// TIA Portal V20 export
// export: Created 2025-12-01T14:57:03.8292158Z, ExportSetting None, DisplayName Totally Integrated Automation Portal, DisplayVersion V20 Update 3, DisplayName TIA Portal Openness, DisplayVersion V20 Update 3, DisplayName TIA Portal Version Control Interface, DisplayVersion V20 Update 3, DisplayName STEP 7 Professional, DisplayVersion V20 Update 3, DisplayName STEP 7 Safety, DisplayVersion V20 Update 2, DisplayName WinCC Basic/Comfort/Advanced, DisplayVersion V20 Update 3, DisplayName WinCC Professional, DisplayVersion V20 Update 3, DisplayName WinCC Unified, DisplayVersion V20 Update 3
FUNCTION "FC702_JDT02RecJdTMensaje" : Void   // FC702, LAD
TITLE = "RecJdTMensaje" Recepción del Mensaje enviado por TCP/IP
{ S7_Optimized_Access := 'FALSE' }
AUTHOR : TRACKING
NAME : 20141014
VERSION : 4.0
// Pasos a seguir, por orden
// 
// - Recoger cabecera
// - Recoger cuerpo
// - Transferir Mensaje recibido por TCP/IP
// stored: AutoNumber false, SetENOAutomatically false
   VAR_TEMP
      DBRecJdt : Word;   // DB de Recpcion de Mensaje
      DBUltimoRec : Word;   // DB del Ultimo Mensaje Recibido
      Longitud : UDInt;   // Longitud del cuerpo
      CantidadBytes : UDInt;   // Cantidad de Bytes de los Eventos
      RecJdT_Longitud : UDInt;   // Longitud de Bytes que recibe en AG_RECV
      ReturnValor : Int;   // Temporal
      POrigen : Any;   // Puntero ANY del Origen
      PDestino : Any;   // Puntero ANY del Destino
   END_VAR
BEGIN

NETWORK
TITLE = Inicializaciones
// -------------------------------------------------------------------------------------------
// Si trabaja sin Agencia  2018 01 24
      SET;
      AN    "Activar_JDT02";  // Mirar si se trabaja con agencia
      JC    Final;

// ------------------------------------------------------------------------------------------------------
// Inicializamos las variables de los DB
      L     "JDT2_NDB_RecMensaje";  // Cogemos el Numero del DB de RecepMensaje
      T     #DBRecJdt;
      L     "JDT2_NDB_UltimoRec";  // Cogemos el Numero del DB de UltimoRecibido
      T     #DBUltimoRec;

// ------------------------------------------------------------------------------------------------------
// Comprobamos el EnlaceCP
      AN    "DB701_JDT02StatusCOM".EnlaceCP_OK;  // Mirar Si esta el EnlaceCP Activo
      JCN   Inicio;

      R     "DB701_JDT02StatusCOM".RecJdT_Cabecera;  // Resetear Variables
      R     "DB701_JDT02StatusCOM".RecJdT_Cuerpo;

      CALL  "FC898_BorrarMensaje"
      ( DB_A_RESET := "DB702_JDT02RecepMensaje"  // ¿Hay que borrarlo?
      );

      JU    Final;  // Finalizar


NETWORK
TITLE = Distribucion
// Orden a mirar para distribucion del trabajo
// - Esta el Cuerpo recogida - Transferir
// - Esta la cabecera recogida - Recoger el Cuerpo
// - Recoger la Cabecera
Inicio:NOP   0;
      SET;
      A     "DB701_JDT02StatusCOM".RecJdT_Cuerpo;  // Esta recogido el Cuerpo
      JC    TranferirMensaje;  // Ir a Transferir el Mensaje

      A     "DB701_JDT02StatusCOM".RecJdT_Cabecera;  // Esta recogido la Cabecera
      JC    RecogerCuerpo;  // Ir a Recoger el Cuerpo

      JU    RecogerCabeza;  // Ir a Recoger la Cabecera



NETWORK
TITLE = Recepcion de la Cabeza del Mensaje
// Pasos a seguir:
// - Generar el Punterp para recoger la Cabecera
// - Mirar si ha llegado la cabecera
// - Comprobación del mensaje recibido es correcto
// - Mirar si hay que resetear el Enlace
// -----------------------------------------------------------------------------------------------------
// 1º Paso - Generar el Puntero para recoger la Cabecera

RecogerCabeza:CALL  "FC897_Generar_PointerAny"
      ( TYP           := 16#10,
        DataTyp       := 16#02,
        repeatcounter := 22,  // Tamaño de la cabecera
        DB_Number     := "JDT2_NDB_RecMensaje",  // DB donde guardar la cabecera
        storearea     := 16#84,
        storeaddresse := 16#0000_0000,
        Any_Pointer   := #POrigen  // Puntero de la cabecera
      );

// -----------------------------------------------------------------------------------------------------
// 2º Paso - Mirar si la llegado la cabecera

      AN    "DB891_VariablesTCP".TRCV_JdT_PLC_Req_JDT02;
      AN    "DB891_VariablesTCP".TRCV_JdT_PLC_Busy_JDT02;
      S     "DB891_VariablesTCP".TRCV_JdT_PLC_Req_JDT02;

      CALL  TRCV, "DB899_TRCV_JdT_PLC_JDT02"
      ( EN_R     := "DB891_VariablesTCP".TRCV_JdT_PLC_Req_JDT02,
        ID       := W#16#3,
        LEN      := 22,
        ADHOC    := ,
        NDR      := "DB891_VariablesTCP".TRCV_JdT_PLC_Done_JDT02,
        BUSY     := "DB891_VariablesTCP".TRCV_JdT_PLC_Busy_JDT02,
        ERROR    := "DB891_VariablesTCP".TRCV_JdT_PLC_Error_JDT02,
        STATUS   := "DB891_VariablesTCP".TRCV_JdT_PLC_Status_JDT02,
        RCVD_LEN := #RecJdT_Longitud,
        DATA     := #POrigen
      );



// -----------------------------------------------------------------------------------------------------
// 3º Paso - Comprobación del mensaje recibido

      A     "DB891_VariablesTCP".TRCV_JdT_PLC_Req_JDT02;  // Si llega el Inicio de Mensaje 0x02
      A     "DB891_VariablesTCP".TRCV_JdT_PLC_Done_JDT02;  // Cabecera ya recogida
      AN    "DB891_VariablesTCP".TRCV_JdT_PLC_Error_JDT02;
      A(;
      L     "DB702_JDT02RecepMensaje".Mensaje[0];
      L     2;
      ==I;
      );
      S     "DB701_JDT02StatusCOM".RecJdT_Cabecera;
      R     "DB891_VariablesTCP".TRCV_JdT_PLC_Req_JDT02;



// -----------------------------------------------------------------------------------------------------
// 4º Paso - Hay que resetear el Enlace

      A     "DB891_VariablesTCP".TRCV_JdT_PLC_Req_JDT02;  // Sino llega el Inicio de Mensaje 0x02
      A     "DB891_VariablesTCP".TRCV_JdT_PLC_Done_JDT02;  // Resetear
      AN    "DB891_VariablesTCP".TRCV_JdT_PLC_Error_JDT02;
      A(;
      L     "DB702_JDT02RecepMensaje".Mensaje[0];
      L     2;
      <>I;
      );
      S     "DB701_JDT02StatusCOM".RecJdT_Reset;
      R     "DB891_VariablesTCP".TRCV_JdT_PLC_Req_JDT02;

      A     "DB891_VariablesTCP".TRCV_JdT_PLC_Req_JDT02;  //Si llega Error en la Recepcio
      AN    "DB891_VariablesTCP".TRCV_JdT_PLC_Done_JDT02;  // Resetear
      A     "DB891_VariablesTCP".TRCV_JdT_PLC_Error_JDT02;
      S     "DB701_JDT02StatusCOM".RecJdT_Reset;
      R     "DB891_VariablesTCP".TRCV_JdT_PLC_Req_JDT02;


//////////////////////////////////////////////////////////////////////////
/// Final (Alonso) 2019 09 19
      SET;
      A     "DB701_JDT02StatusCOM".RecJdT_Cabecera;
      JC    RecogerCuerpo;

      JU    Final;  // Finalizar



NETWORK
TITLE = Recepcion del Cuerpo del Mensaje
// Pasos a seguir
// - Conseguir la longitud del cuerpo
// - Generar el puntero para recoger el cuerpo
// - Mirar si ha llegado el cuerpo
// - Comprobación del mensaje recibido es correcto
// - Mirar si hay que resetear el Enlace
// -----------------------------------------------------------------------------------------------------
// 1º Paso - Conseguir la longitud del cuerpo
RecogerCuerpo:CALL  "FC890_EtiqChar_EtiqDInt"
      ( DB_String   := "JDT2_NDB_RecMensaje",
        Long_String := 5,
        Offset_Ini  := 20,
        Valor       := #Longitud
      );  // Conseguir del Mensaje su longitud

      L     #Longitud;
      T     "DB701_JDT02StatusCOM".RecJdT_LongitudCuerpo;  // Guardo la longitud del Mensaje

      L     "DB701_JDT02StatusCOM".RecJdT_LongitudCuerpo;  // Calculo la longitud del Cuerpo
      L     22;
      -I;
      T     #CantidadBytes;


// -----------------------------------------------------------------------------------------------------
// 2º Paso - Generar el Puntero para recoger la Cuerpo
      CALL  "FC897_Generar_PointerAny"
      ( TYP           := 16#10,
        DataTyp       := 16#02,
        repeatcounter := #CantidadBytes,  // Tamaño del cuerpo
        DB_Number     := "JDT2_NDB_RecMensaje",  // DB donde guardar el cuerpo
        storearea     := 16#84,
        storeaddresse := 16#0000_00B0,  // Adress Byte 22 Bit 0 -> Hex:B0
        Any_Pointer   := #POrigen  // Puntero del cuerpo
      );

// -----------------------------------------------------------------------------------------------------
// 2º Paso - Mirar si la llegado el cuerpo



      AN    "DB891_VariablesTCP".TRCV_JdT_PLC_Req_JDT02;
      AN    "DB891_VariablesTCP".TRCV_JdT_PLC_Busy_JDT02;
      S     "DB891_VariablesTCP".TRCV_JdT_PLC_Req_JDT02;

      CALL  TRCV, "DB899_TRCV_JdT_PLC_JDT02"
      ( EN_R     := "DB891_VariablesTCP".TRCV_JdT_PLC_Req_JDT02,
        ID       := W#16#3,
        LEN      := #CantidadBytes,
        ADHOC    := ,
        NDR      := "DB891_VariablesTCP".TRCV_JdT_PLC_Done_JDT02,
        BUSY     := "DB891_VariablesTCP".TRCV_JdT_PLC_Busy_JDT02,
        ERROR    := "DB891_VariablesTCP".TRCV_JdT_PLC_Error_JDT02,
        STATUS   := "DB891_VariablesTCP".TRCV_JdT_PLC_Status_JDT02,
        RCVD_LEN := #RecJdT_Longitud,
        DATA     := #POrigen
      );




// -----------------------------------------------------------------------------------------------------
// 3º Paso - Comprobación del mensaje recibido

      A     "DB891_VariablesTCP".TRCV_JdT_PLC_Req_JDT02;  // Comprobar si ha llegado el cuerpo
      A     "DB891_VariablesTCP".TRCV_JdT_PLC_Done_JDT02;
      AN    "DB891_VariablesTCP".TRCV_JdT_PLC_Error_JDT02;
      S     "DB701_JDT02StatusCOM".RecJdT_Cuerpo;
      R     "DB891_VariablesTCP".TRCV_JdT_PLC_Req_JDT02;



// -----------------------------------------------------------------------------------------------------
// 4º Paso - Hay que resetear el Enlace

      A     "DB891_VariablesTCP".TRCV_JdT_PLC_Req_JDT02;  //Si llega Error en la Recepcion
      AN    "DB891_VariablesTCP".TRCV_JdT_PLC_Done_JDT02;  // Resetear
      A     "DB891_VariablesTCP".TRCV_JdT_PLC_Error_JDT02;
      S     "DB701_JDT02StatusCOM".RecJdT_Reset;
      R     "DB891_VariablesTCP".TRCV_JdT_PLC_Req_JDT02;


//////////////////////////////////////////////////////////////////////////
/// Final (Alonso) 2019 09 19
      SET;
      A     "DB701_JDT02StatusCOM".RecJdT_Cuerpo;
      JC    TranferirMensaje;

      JU    Final;  // Finalizar


NETWORK
TITLE = Transferencia del Mensaje Recibido por TCP/IP
// Pasos a sefuir:
// - Calcular los punteros Origen y destino
// - Transferir
// - Resetear las variables internas
TranferirMensaje:L     0;  // Mirar si se puede transferir ya
      LAR1;
      OPN   DB [#DBUltimoRec];
      L     DBB [AR1, P#0.0];
      L     0;
      <>I;
      JC    Final;

// -----------------------------------------------------------------------------------------------------
// 1º Paso - Calcular los Puntero Origen y Destino
      L     "DB701_JDT02StatusCOM".RecJdT_LongitudCuerpo;  // Calculo la longitud del Cuerpo
      T     #CantidadBytes;

      CALL  "FC897_Generar_PointerAny"
      ( TYP           := 16#10,
        DataTyp       := 16#02,
        repeatcounter := #CantidadBytes,  // Tamaño del mensaje
        DB_Number     := "JDT2_NDB_RecMensaje",  // DB fuente
        storearea     := 16#84,
        storeaddresse := 16#0000_0000,
        Any_Pointer   := #POrigen  // Puntero del UltimoRecibido
      );

      CALL  "FC897_Generar_PointerAny"
      ( TYP           := 16#10,
        DataTyp       := 16#02,
        repeatcounter := #CantidadBytes,  // Tamaño del mensaje
        DB_Number     := "JDT2_NDB_UltimoRec",  // DB donde guardar el UltimoRecibido
        storearea     := 16#84,
        storeaddresse := 16#0000_0000,
        Any_Pointer   := #PDestino  // Puntero del UltimoRecibido
      );

// -----------------------------------------------------------------------------------------------------
// 2º Paso - Transferir
      CALL  BLKMOV
      ( SRCBLK  := #POrigen,
        RET_VAL := #ReturnValor,
        DSTBLK  := #PDestino
      );

// -----------------------------------------------------------------------------------------------------
// 3º Paso - Resetear variables internas
      SET;
      R     "DB701_JDT02StatusCOM".RecJdT_Cabecera;  // Resetear Variables
      R     "DB701_JDT02StatusCOM".RecJdT_Cuerpo;
      CALL  "FC898_BorrarMensaje"
      ( DB_A_RESET := "DB702_JDT02RecepMensaje"  // ¿Hay que borrarlo todo?
      );

      JU    Final;  // Finalizar


NETWORK
TITLE = Finalizar la funcion
// - Se Acabo la Función
Final:NOP   0;

END_FUNCTION
